FUNCTION_BLOCK FB_Auto_PC
VAR_INPUT
	bEnable				: BOOL;
END_VAR	
VAR_OUTPUT
	fPCV				: LREAL;
	fSCV				: LREAL;

END_VAR
VAR
	//Function Blocks
	fbAutoStartPos		: FB_AutoStartPos;
	fbAutoSineMotion	: FB_AutoSineMotion;
	
	fbClock				: FB_Clock;
	
	bStartPosOK			: BOOL;

END_VAR
VAR // added by the converter: edge detectors and wires of the graphical bodies
    _w1 : LREAL;
END_VAR

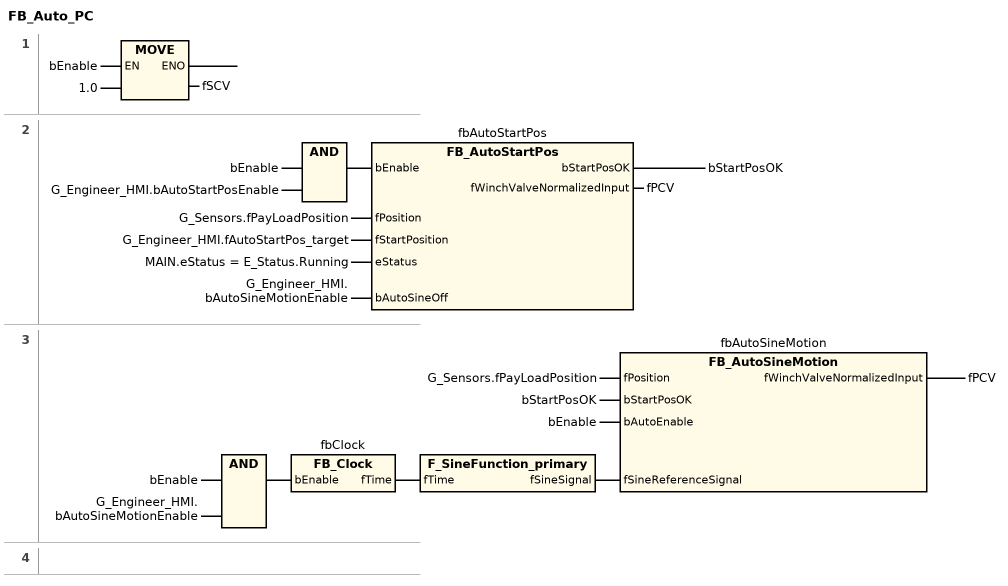
// NETWORK 1
IF bEnable THEN fSCV := 1.0; END_IF

// NETWORK 2
fbAutoStartPos(
    bEnable := bEnable AND G_Engineer_HMI.bAutoStartPosEnable,
    fPosition := G_Sensors.fPayLoadPosition,
    fStartPosition := G_Engineer_HMI.fAutoStartPos_target,
    eStatus := MAIN.eStatus = E_Status.Running,
    bAutoSineOff := G_Engineer_HMI.bAutoSineMotionEnable,
    fWinchValveNormalizedInput => fPCV); // FB_AutoStartPos
bStartPosOK := fbAutoStartPos.bStartPosOK;

// NETWORK 3
fbClock(bEnable := bEnable AND G_Engineer_HMI.bAutoSineMotionEnable); // FB_Clock
F_SineFunction_primary(fTime := fbClock.fTime, fSineSignal => _w1);
fbAutoSineMotion(
    fPosition := G_Sensors.fPayLoadPosition,
    bStartPosOK := bStartPosOK,
    bAutoEnable := bEnable,
    fSineReferenceSignal := _w1); // FB_AutoSineMotion
fPCV := fbAutoSineMotion.fWinchValveNormalizedInput;

// NETWORK 4

END_FUNCTION_BLOCK

(* stored: Version 1.1.0.1
   POU FB_Auto_PC: Id {08676a61-e483-474a-90df-258b50adcd27}, SpecialFunc None *)
